TYPE ST_LCP1_Base :
STRUCT
	Segment	: ARRAY [1..3] OF ST_Segment_Base;
		
	Segment1to3_ShortContactClose	: BOOL;
	Segment1to3_UnShortContactClose	: BOOL;
	Segment4to6_ShortContactClose	: BOOL;
	Segment4to6_UnShortContactClose	: BOOL;
	LossInterlockPressure			: BOOL;
	PSU1OK							: BOOL;
	
	Fire			: BOOL;
	SegmentCharged	: BOOL;
	TriggerScope	: BOOL;
END_STRUCT
END_TYPE

(* stored: Version 1.1.0.1, ProductVersion 3.1.4024.11
   DUT ST_LCP1_Base: Id {ae8b38a8-6b87-473a-a194-b814e6159583} *)
